FUNCTION_BLOCK Average
VAR_INPUT
	NewSample: LREAL;
END_VAR
VAR_OUTPUT
	Value: LREAL;
END_VAR
VAR
	Acc: lreal;
	LastSec: LINT;
END_VAR

IF LastSec = 0 THEN
	Acc := NewSample;
END_IF
IF Globals.SecondsCounter <> LastSec THEN
	Acc := Acc * 0.9;
	Acc := Acc + NewSample;
	Value := Acc / 10;
	LastSec := Globals.SecondsCounter;
END_IF

END_FUNCTION_BLOCK

(* stored: Version 1.1.0.1, ProductVersion 3.1.4024.4
   POU Average: Id {b5d1a686-8d96-4aa9-ad7b-e544505a4d3d}, SpecialFunc None *)
